{attribute addProperty BoxType "EK1100-0000-0018"}
{attribute addProperty Id "TcTerminals210_1BK1250TcTerminals210_1BK1250_5A51D77700"}
{attribute addProperty CRC "2568560333"}
{attribute addProperty SizeInBites "0"}
{attribute addProperty SizeInBytes "0"}
TYPE TcTerminals210_EK1100_1_99191ECD EXTENDS EK1100_179A0949 :
STRUCT
	{attribute addProperty Name "TcTerminals210_1BK1250"}
	TcTerminals210_1BK1250 : TcTerminals210_1BK1250_5A51D777;
END_STRUCT
END_TYPE

(* stored: Version 1.2.0.0, ProductVersion 3.1.4024.9
   DUT TcTerminals210_EK1100_1_99191ECD: Id {be33d3d4-6c6c-4598-adea-7f4a435c7570} *)
